FUNCTION F_Concat4_Large : LongString
VAR_IN_OUT CONSTANT
   sOne : LongString;
   sTwo : LongString;
   sThree : LongString;
   sFour : LongString;
END_VAR
VAR
   str : LongString;
END_VAR

str := F_Concat3_Large(sTwo, sThree, sFour);

F_Concat4_Large :=
   F_ConcatLarge(
      sOne,
      str
   );

END_FUNCTION

(* stored: Version 1.1.0.1, ProductVersion 3.1.4024.9
   POU F_Concat4_Large: Id {7fff765e-4441-481f-8fdf-a597e0aec267}, SpecialFunc None *)
